SUBAPPLICATION PAGES (* Subapplication Type *)
  (* Standard: 61499-2 *)
  (* Version 1.0, 2023-02-06, franz *)
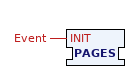
  EVENT_INPUT
    INIT;
  END_EVENT
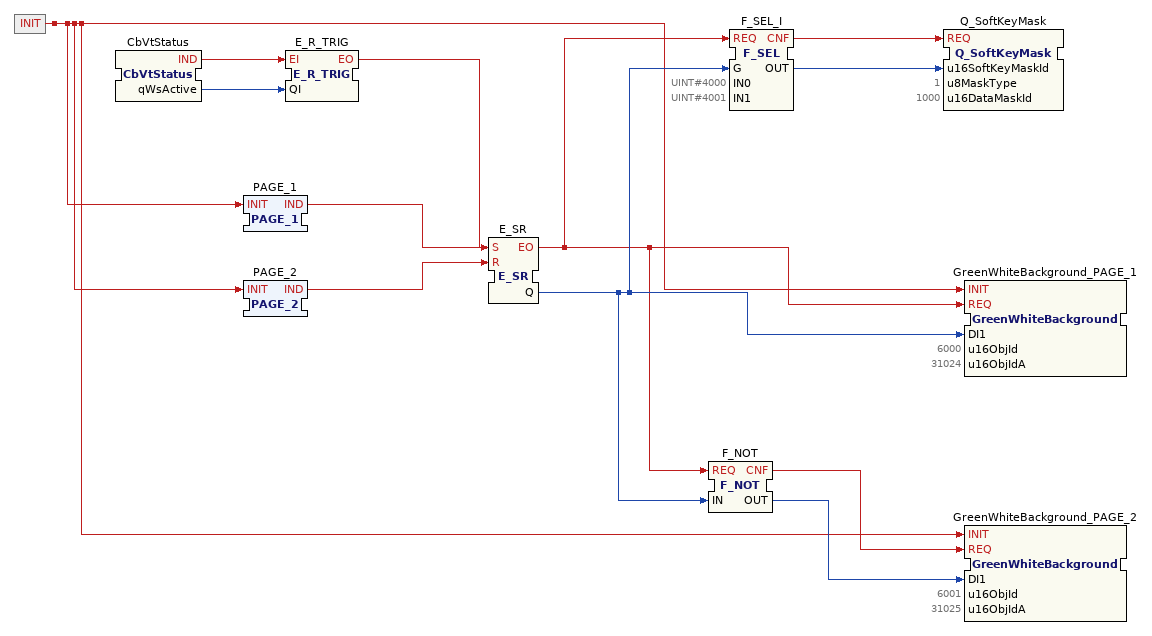
  FBS
    GreenWhiteBackground_PAGE_1 : GreenWhiteBackground(u16ObjId := 6000, u16ObjIdA := 31024);
    GreenWhiteBackground_PAGE_2 : GreenWhiteBackground(u16ObjId := 6001, u16ObjIdA := 31025);
    E_SR : E_SR;
    F_NOT : F_NOT;
    Q_SoftKeyMask : Q_SoftKeyMask(u8MaskType := 1, u16DataMaskId := 1000);
    F_SEL_I : F_SEL(IN0 := UINT#4000, IN1 := UINT#4001);
    CbVtStatus : CbVtStatus;
    E_R_TRIG : E_R_TRIG;
  END_FBS
  SUBAPPS
    PAGE_1 : PAGE_1;
    PAGE_2 : PAGE_2;
  END_SUBAPPS
  EVENT_CONNECTIONS
    INIT TO GreenWhiteBackground_PAGE_1.INIT;
    INIT TO PAGE_1.INIT;
    INIT TO PAGE_2.INIT;
    INIT TO GreenWhiteBackground_PAGE_2.INIT;
    PAGE_1.IND TO E_SR.S;
    PAGE_2.IND TO E_SR.R;
    E_SR.EO TO F_NOT.REQ;
    E_SR.EO TO GreenWhiteBackground_PAGE_1.REQ;
    F_NOT.CNF TO GreenWhiteBackground_PAGE_2.REQ;
    E_SR.EO TO F_SEL_I.REQ;
    F_SEL_I.CNF TO Q_SoftKeyMask.REQ;
    CbVtStatus.IND TO E_R_TRIG.EI;
    E_R_TRIG.EO TO E_SR.S;
  END_CONNECTIONS
  DATA_CONNECTIONS
    E_SR.Q TO GreenWhiteBackground_PAGE_1.DI1;
    E_SR.Q TO F_NOT.IN;
    F_NOT.OUT TO GreenWhiteBackground_PAGE_2.DI1;
    F_SEL_I.OUT TO Q_SoftKeyMask.u16SoftKeyMaskId;
    E_SR.Q TO F_SEL_I.G;
    CbVtStatus.qWsActive TO E_R_TRIG.QI;
  END_CONNECTIONS
END_SUBAPPLICATION
